(* CODESYS project EtherNetIPServices_Example.project
   Title: EtherNet IP Services Example
   Description: An example project of how to use the EtherNet/IP Services library.

Project tree, tasks and I/O mapping:
  Device : CODESYS Control Win V3 x64, 3S - Smart Software Solutions GmbH, version 3.5.14.0
    application Application
      libraries: Standard, 3.5.14.0 (System)
      task MainTask (cyclic, interval t#20ms, priority 1) calls PLC_PRG
      program PLC_PRG [ST]
      data type STRING64
      license
    Ethernet : Ethernet, 3S - Smart Software Solutions GmbH, version 3.5.14.0
        settings: NetworkInterfaceName = 'ether0'
      EtherNet_IP_Scanner : EtherNet/IP Scanner, 3S - Smart Software Solutions GmbH, order no. 1, version 3.5.14.0
        _1734_AENT_Ethernet_Adapter : 1734-AENT Ethernet Adapter, Allen-Bradley Company, Inc., order no. 1734-AENT, version Major Revision=16#3, Minor Revision = 16#1
            settings: INITIALIZED = TRUE; IP address of Target = [16#C0,16#A8,16#01,16#02]; Keying.Check Minor Revision = FALSE
        WAGO_750_352_FC_ETHERNET : WAGO 750-352 FC ETHERNET, Wago Kontakttechnik, order no. 750-352, version Major Revision=16#1, Minor Revision = 16#1
            settings: INITIALIZED = TRUE; IP address of Target = [16#C0,16#A8,16#01,16#05]; Keying.Check Minor Revision = FALSE
        Generic_EthernetIP_device : Generic EthernetIP device, 3S - Smart Software Solutions GmbH, version 3.4.2.0
            settings: INITIALIZED = TRUE; IP address of Target = [16#C0,16#A8,16#01,16#04]
  00000000-0000-0000-0000-000000000000|C:\Users\m.lamp\Documents\license.txt
*)

// Device/Application/STRING64
(* CIP Data type for string with a length of max. 64 chars *)
TYPE STRING64 :
STRUCT
	uiLength	: UINT;
	sString		: STRING(63);
END_STRUCT
END_TYPE

// Device/Application/PLC_PRG
PROGRAM PLC_PRG
VAR
	reset				: ENIP.Reset;					(* fb to reset a cip class *)
	getAttributeSingle	: ENIP.Get_Attribute_Single;	(* fb to get a single attribute from a cip class *)
	setAttributeSingle	: ENIP.Set_Attribute_Single;	(* fb to set a single attribute of a cip class *)
	udiReceivedData		: UDINT;						
	strHostnameToSet	: STRING64 := (sString := 'NewName');		
	strHostnameToGet	: STRING64;		
END_VAR

(* this instance call requests the host name (= name of the device in the network) from the WAGO_750_352_FC_ETHERNET device as soon as xExecute gets TRUE *)
getAttributeSingle(
	xExecute:= , 
	itfEtherNetIPDevice:= WAGO_750_352_FC_ETHERNET, 	(* instance of the device (instance is found in the I/O Image of the device) *)
	eClass:= ENIP.CIPClass.TCPIPInterfaceObject,		(* cip class which contains the desired attribute *)
	dwInstance:= 1, 									(* value of 0 is class level, range from 1..x is instance level *)
	pData:= ADR(strHostnameToGet),						(* data buffer *)
	udiDataSize:= SIZEOF(strHostnameToGet), 			(* size of the data buffer *)
	wAttribute:= 6,									(* attribute no. 6 of the tcp/ip interface object is the Hostname (CIP Spec. Vol.2 Chapter 5-3.3.2.6)*)	 
	xDone=> , 
	xBusy=> , 
	xError=> , 
	eError=> , 
	udiReceivedDataSize=> udiReceivedData);				(* if the request was successfull, udiReceivedData contains the number of bytes which have been received *)
	
(* this instance call sets the host name of the WAGO_750_352_FC_ETHERNET as soon as xExecute gets TRUE *)
strHostnameToSet.uiLength := INT_TO_UINT(Standard.LEN(strHostnameToSet.sString));
setAttributeSingle(
	xExecute:= , 
	itfEtherNetIPDevice:= WAGO_750_352_FC_ETHERNET, 	(* instance of the device (instance is found in the I/O Image of the device) *)
	eClass:= ENIP.CIPClass.TCPIPInterfaceObject,        (* cip class which contains the desired attribute *)
	dwInstance:= 1,                                    (* value of 0 is class level, range from 1..x is instance level *)
	pData:= ADR(strHostnameToSet), 						(* data to be assigned to the attribute *)
	udiDataSize:= SIZEOF(strHostnameToSet.uiLength) + strHostnameToSet.uiLength, (* size of the data. Here: size of the Length-Parameter PLUS the length of the string *)
	wAttribute:= 6, 									(* attribute no. 6 of the tcp/ip interface object is the Hostname (CIP Spec. Vol.2 Chapter 5-3.3.2.6)*)	
	xDone=> , 
	xBusy=> , 
	xError=> , 
	eError=> );
	
(* this instance call resets the WAGO_750_352_FC_ETHERNET device as soon as xExecute gets TRUE *)
reset(
	xExecute:= , 
	itfEtherNetIPDevice:= WAGO_750_352_FC_ETHERNET, 	(* instance of the device (instance is found in the I/O Image of the device) *)
	eClass:= ENIP.CIPClass.IdentityObject,              (* cip class which contains the desired attribute *)
	dwInstance:= 1,                                    (* value of 0 is class level, range from 1..x is instance level *)
	xDone=> , 
	xBusy=> , 
	xError=> , 
	eError=> );

END_PROGRAM
